(* Logix 5000 project; controller Sucrose_Main Emulate 5570 rev 20.12; software revision 20.01; part 17 of 30 *)
(* tags used below, declared in another part *)
   Alarm_ACK_Master_Timer : TIMER;
   DO_E22_5 : ALIAS FOR FLX_E22:5:O;   // Discrete Output EN2T_FLX 192.168.1.22
   FV230602_AOI : QSI_Flow_Valve;   // FV-23-06-02 PRE FILTER TRAIN 2 INLET LOW POINT DRAIN VALVE
   FV230603_AOI : QSI_Flow_Valve;   // FV-23-06-03 PRE FILTER TRAIN 2 INLET LOW POINT DRAIN VALVE
   FV230604_AOI : QSI_Flow_Valve;   // FV-23-06-04 PRE FILTER TRAIN 2 OUTLET LOW POINT DRAIN VALVE
   FV230605_AOI : QSI_Flow_Valve;   // FV-23-06-05 PRE FILTER TRAIN 2 OUTLET LOW POINT DRAIN VALVE
   FV230607_AOI : QSI_Flow_Valve;   // FV-23-06-07 LOW POINT DRAIN VALVE
   FV230609_AOI : QSI_Flow_Valve;   // FV-23-06-09 FINAL FILTER TRAIN 2 INLET LOW POINT DRAIN VALVE
   FV230610_AOI : QSI_Flow_Valve;   // FV-23-06-10 FINAL FILTER TRAIN 2 INLET LOW POINT DRAIN VALVE
   FV230611_AOI : QSI_Flow_Valve;   // FV-23-06-11 FINAL FILTER TRAIN 2 OUTLET LOW POINT DRAIN VALVE
   FV230612_AOI : QSI_Flow_Valve;   // FV-23-06-12 FINAL FILTER TRAIN 2 OUTLET LOW POINT DRAIN VALVE
   Sucrose_MM_Enable : BOOL;
   SucroseCIP_FILTRATION_REMOTE : CIP_REMOTE;
   SucroseFiltration : Area_Program;
(* FiltrationArea_EN2T_IO_Discrete_DO_E22_5, continued *)

ROUTINE _03_FV230602   (* ladder *)
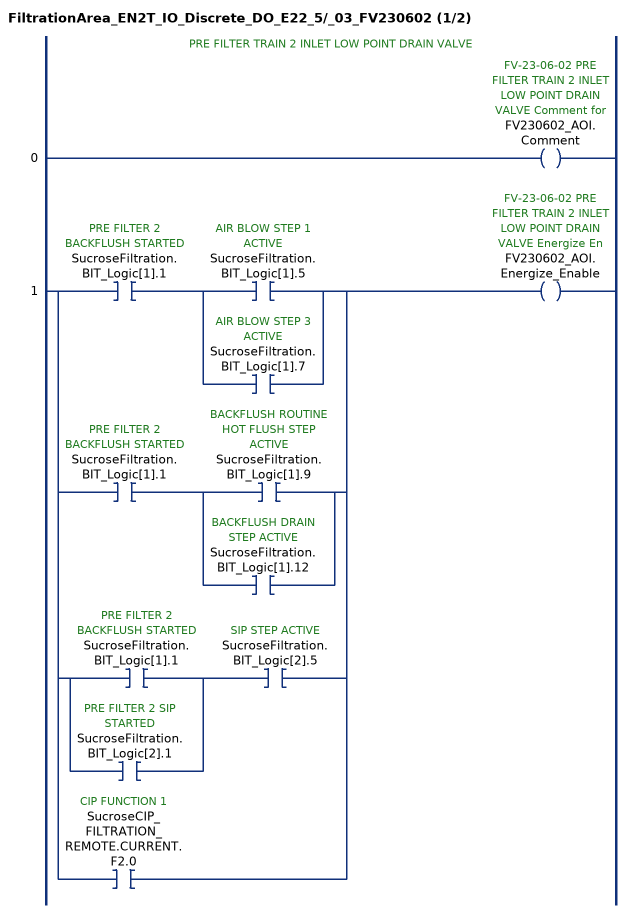
   // PRE FILTER TRAIN 2 INLET LOW POINT DRAIN VALVE
   0: OTE(FV230602_AOI.Comment);
   1: [XIC(SucroseFiltration.BIT_Logic[1].1) [XIC(SucroseFiltration.BIT_Logic[1].5) ,XIC(SucroseFiltration.BIT_Logic[1].7) ] ,XIC(SucroseFiltration.BIT_Logic[1].1) [XIC(SucroseFiltration.BIT_Logic[1].9) ,XIC(SucroseFiltration.BIT_Logic[1].12) ] ,[XIC(SucroseFiltration.BIT_Logic[1].1) ,XIC(SucroseFiltration.BIT_Logic[2].1) ] XIC(SucroseFiltration.BIT_Logic[2].5) ,XIC(SucroseCIP_FILTRATION_REMOTE.CURRENT.F2.0) ]OTE(FV230602_AOI.Energize_Enable);
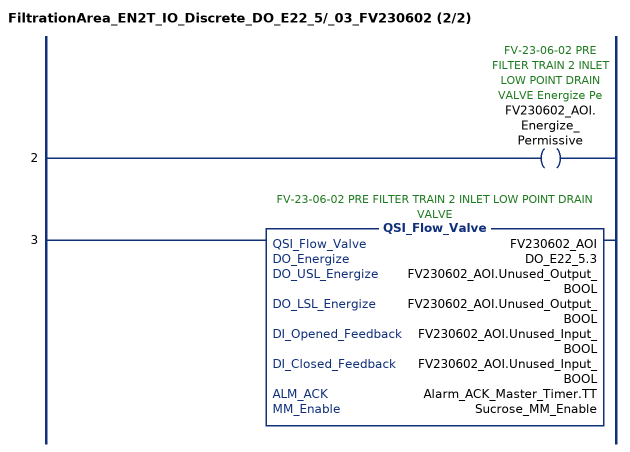
   2: OTE(FV230602_AOI.Energize_Permissive);
   3: QSI_Flow_Valve(FV230602_AOI,DO_E22_5.3,FV230602_AOI.Unused_Output_BOOL,FV230602_AOI.Unused_Output_BOOL,FV230602_AOI.Unused_Input_BOOL,FV230602_AOI.Unused_Input_BOOL,Alarm_ACK_Master_Timer.TT,Sucrose_MM_Enable);
END_ROUTINE

ROUTINE _04_FV230603   (* ladder *)
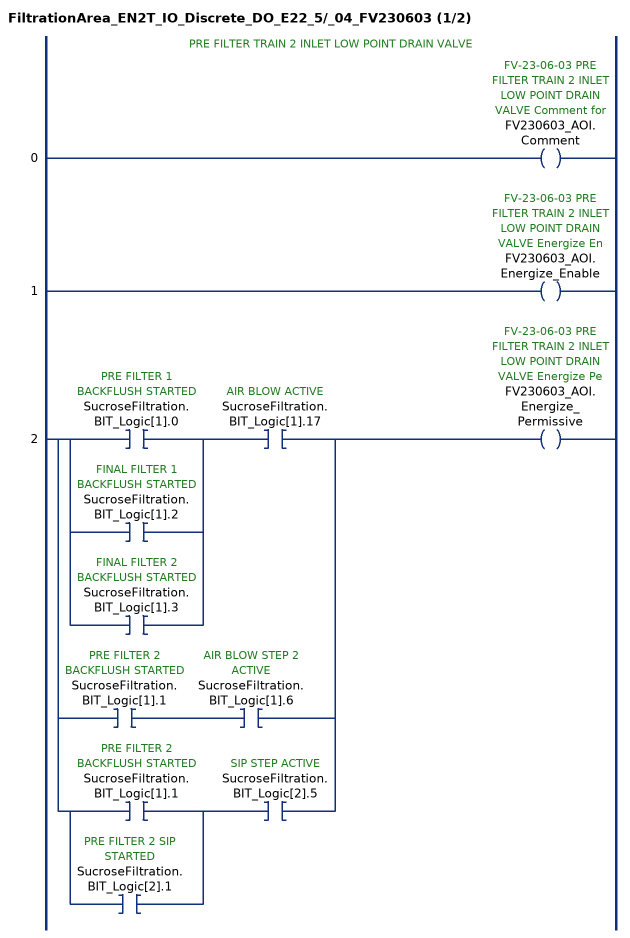
   // PRE FILTER TRAIN 2 INLET LOW POINT DRAIN VALVE
   0: OTE(FV230603_AOI.Comment);
   1: OTE(FV230603_AOI.Energize_Enable);
   2: [[XIC(SucroseFiltration.BIT_Logic[1].0) ,XIC(SucroseFiltration.BIT_Logic[1].2) ,XIC(SucroseFiltration.BIT_Logic[1].3) ] XIC(SucroseFiltration.BIT_Logic[1].17) ,XIC(SucroseFiltration.BIT_Logic[1].1) XIC(SucroseFiltration.BIT_Logic[1].6) ,[XIC(SucroseFiltration.BIT_Logic[1].1) ,XIC(SucroseFiltration.BIT_Logic[2].1) ] XIC(SucroseFiltration.BIT_Logic[2].5) ]OTE(FV230603_AOI.Energize_Permissive);
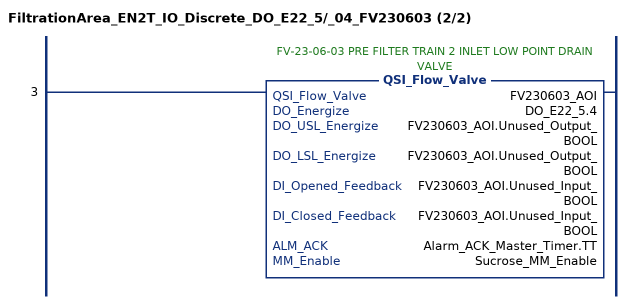
   3: QSI_Flow_Valve(FV230603_AOI,DO_E22_5.4,FV230603_AOI.Unused_Output_BOOL,FV230603_AOI.Unused_Output_BOOL,FV230603_AOI.Unused_Input_BOOL,FV230603_AOI.Unused_Input_BOOL,Alarm_ACK_Master_Timer.TT,Sucrose_MM_Enable);
END_ROUTINE

ROUTINE _05_FV230604   (* ladder *)
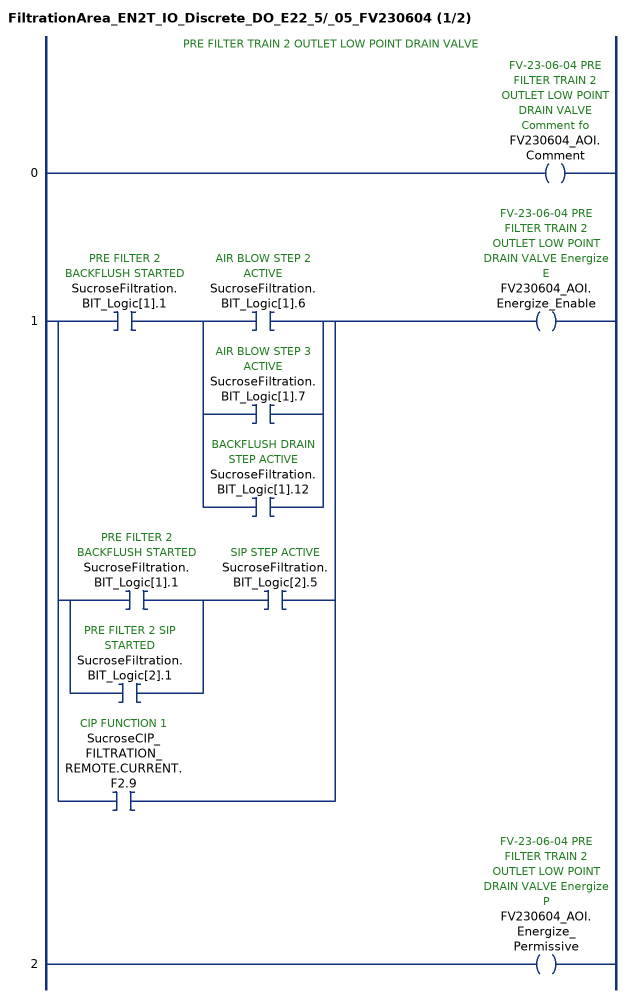
   // PRE FILTER TRAIN 2 OUTLET LOW POINT DRAIN VALVE
   0: OTE(FV230604_AOI.Comment);
   1: [XIC(SucroseFiltration.BIT_Logic[1].1) [XIC(SucroseFiltration.BIT_Logic[1].6) ,XIC(SucroseFiltration.BIT_Logic[1].7) ,XIC(SucroseFiltration.BIT_Logic[1].12) ] ,[XIC(SucroseFiltration.BIT_Logic[1].1) ,XIC(SucroseFiltration.BIT_Logic[2].1) ] XIC(SucroseFiltration.BIT_Logic[2].5) ,XIC(SucroseCIP_FILTRATION_REMOTE.CURRENT.F2.9) ]OTE(FV230604_AOI.Energize_Enable);
   2: OTE(FV230604_AOI.Energize_Permissive);
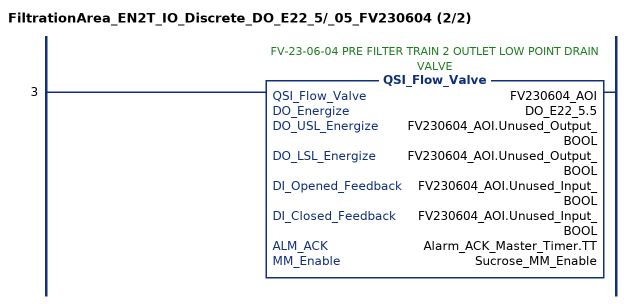
   3: QSI_Flow_Valve(FV230604_AOI,DO_E22_5.5,FV230604_AOI.Unused_Output_BOOL,FV230604_AOI.Unused_Output_BOOL,FV230604_AOI.Unused_Input_BOOL,FV230604_AOI.Unused_Input_BOOL,Alarm_ACK_Master_Timer.TT,Sucrose_MM_Enable);
END_ROUTINE

ROUTINE _06_FV230605   (* ladder *)
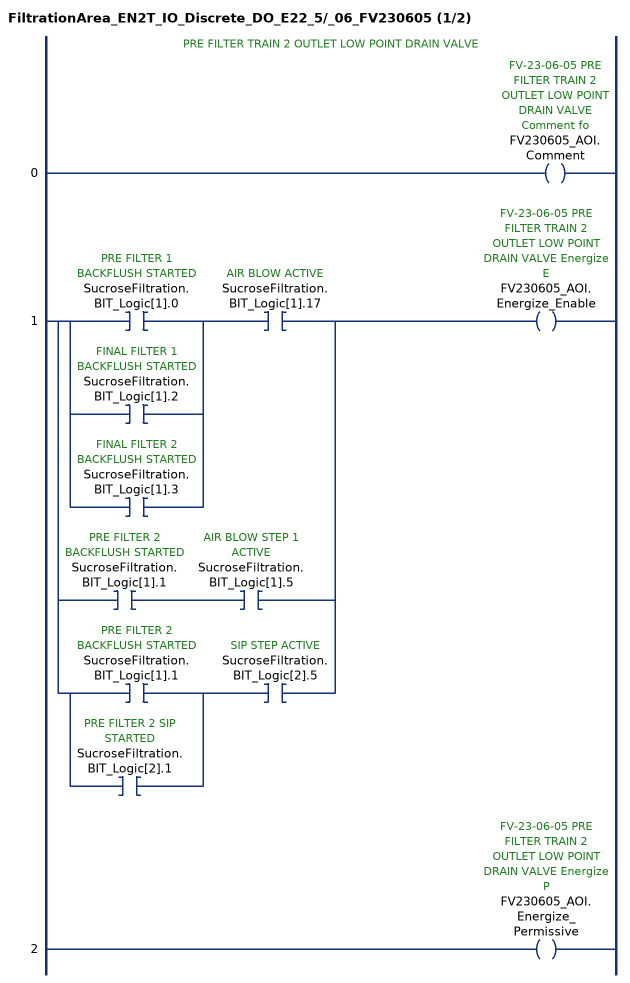
   // PRE FILTER TRAIN 2 OUTLET LOW POINT DRAIN VALVE
   0: OTE(FV230605_AOI.Comment);
   1: [[XIC(SucroseFiltration.BIT_Logic[1].0) ,XIC(SucroseFiltration.BIT_Logic[1].2) ,XIC(SucroseFiltration.BIT_Logic[1].3) ] XIC(SucroseFiltration.BIT_Logic[1].17) ,XIC(SucroseFiltration.BIT_Logic[1].1) XIC(SucroseFiltration.BIT_Logic[1].5) ,[XIC(SucroseFiltration.BIT_Logic[1].1) ,XIC(SucroseFiltration.BIT_Logic[2].1) ] XIC(SucroseFiltration.BIT_Logic[2].5) ]OTE(FV230605_AOI.Energize_Enable);
   2: OTE(FV230605_AOI.Energize_Permissive);
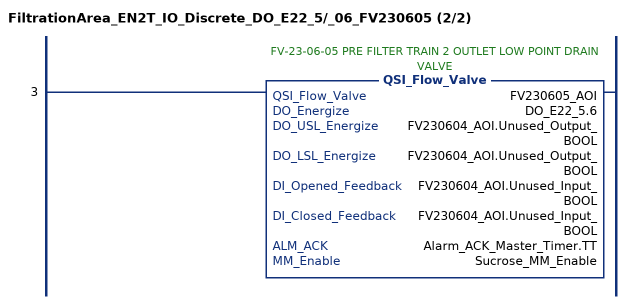
   3: QSI_Flow_Valve(FV230605_AOI,DO_E22_5.6,FV230604_AOI.Unused_Output_BOOL,FV230604_AOI.Unused_Output_BOOL,FV230604_AOI.Unused_Input_BOOL,FV230604_AOI.Unused_Input_BOOL,Alarm_ACK_Master_Timer.TT,Sucrose_MM_Enable);
END_ROUTINE

ROUTINE _07_FV230607   (* ladder *)
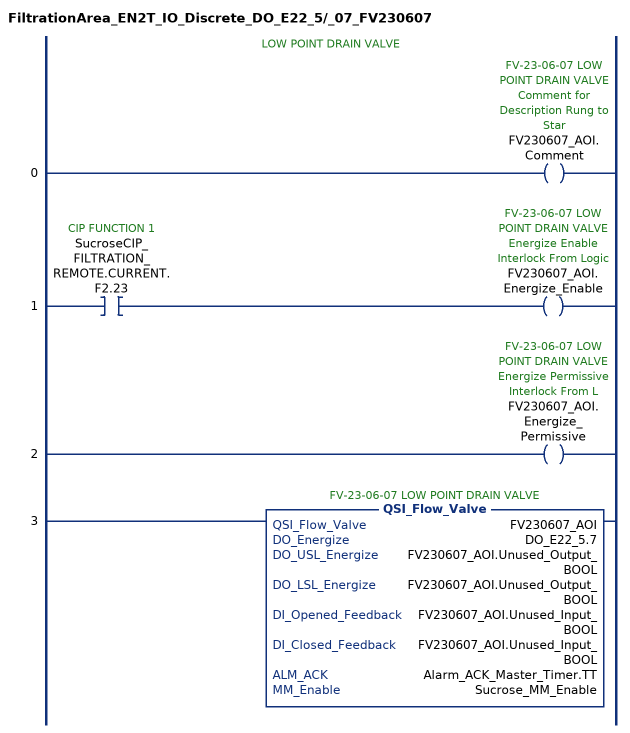
   // LOW POINT DRAIN VALVE
   0: OTE(FV230607_AOI.Comment);
   1: XIC(SucroseCIP_FILTRATION_REMOTE.CURRENT.F2.23)OTE(FV230607_AOI.Energize_Enable);
   2: OTE(FV230607_AOI.Energize_Permissive);
   3: QSI_Flow_Valve(FV230607_AOI,DO_E22_5.7,FV230607_AOI.Unused_Output_BOOL,FV230607_AOI.Unused_Output_BOOL,FV230607_AOI.Unused_Input_BOOL,FV230607_AOI.Unused_Input_BOOL,Alarm_ACK_Master_Timer.TT,Sucrose_MM_Enable);
END_ROUTINE

ROUTINE _08_FV230609   (* ladder *)
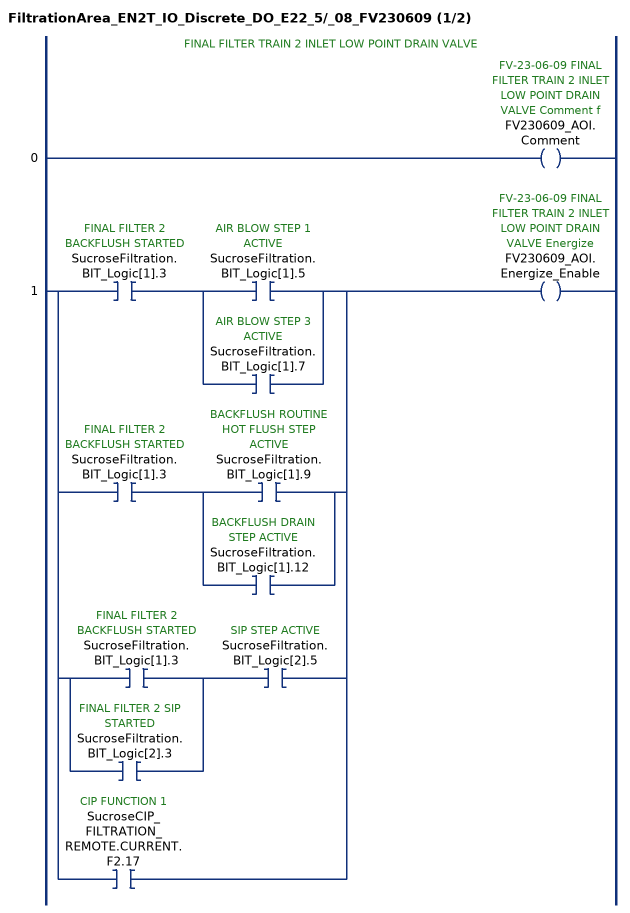
   // FINAL FILTER TRAIN 2 INLET LOW POINT DRAIN VALVE
   0: OTE(FV230609_AOI.Comment);
   1: [XIC(SucroseFiltration.BIT_Logic[1].3) [XIC(SucroseFiltration.BIT_Logic[1].5) ,XIC(SucroseFiltration.BIT_Logic[1].7) ] ,XIC(SucroseFiltration.BIT_Logic[1].3) [XIC(SucroseFiltration.BIT_Logic[1].9) ,XIC(SucroseFiltration.BIT_Logic[1].12) ] ,[XIC(SucroseFiltration.BIT_Logic[1].3) ,XIC(SucroseFiltration.BIT_Logic[2].3) ] XIC(SucroseFiltration.BIT_Logic[2].5) ,XIC(SucroseCIP_FILTRATION_REMOTE.CURRENT.F2.17) ]OTE(FV230609_AOI.Energize_Enable);
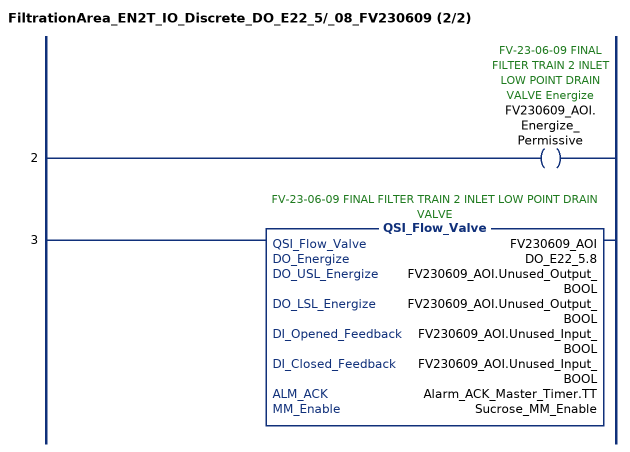
   2: OTE(FV230609_AOI.Energize_Permissive);
   3: QSI_Flow_Valve(FV230609_AOI,DO_E22_5.8,FV230609_AOI.Unused_Output_BOOL,FV230609_AOI.Unused_Output_BOOL,FV230609_AOI.Unused_Input_BOOL,FV230609_AOI.Unused_Input_BOOL,Alarm_ACK_Master_Timer.TT,Sucrose_MM_Enable);
END_ROUTINE

ROUTINE _09_FV230610   (* ladder *)
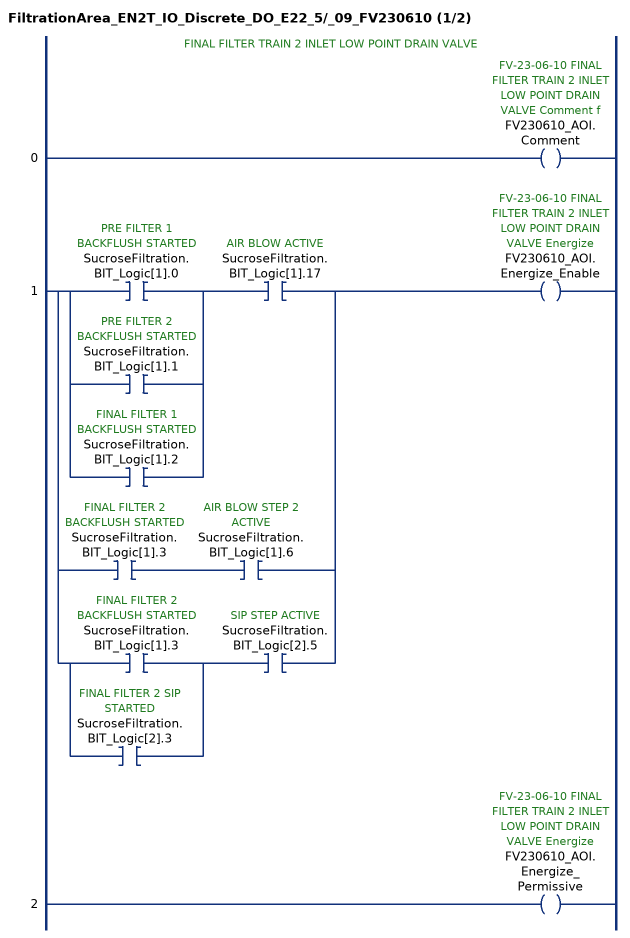
   // FINAL FILTER TRAIN 2 INLET LOW POINT DRAIN VALVE
   0: OTE(FV230610_AOI.Comment);
   1: [[XIC(SucroseFiltration.BIT_Logic[1].0) ,XIC(SucroseFiltration.BIT_Logic[1].1) ,XIC(SucroseFiltration.BIT_Logic[1].2) ] XIC(SucroseFiltration.BIT_Logic[1].17) ,XIC(SucroseFiltration.BIT_Logic[1].3) XIC(SucroseFiltration.BIT_Logic[1].6) ,[XIC(SucroseFiltration.BIT_Logic[1].3) ,XIC(SucroseFiltration.BIT_Logic[2].3) ] XIC(SucroseFiltration.BIT_Logic[2].5) ]OTE(FV230610_AOI.Energize_Enable);
   2: OTE(FV230610_AOI.Energize_Permissive);
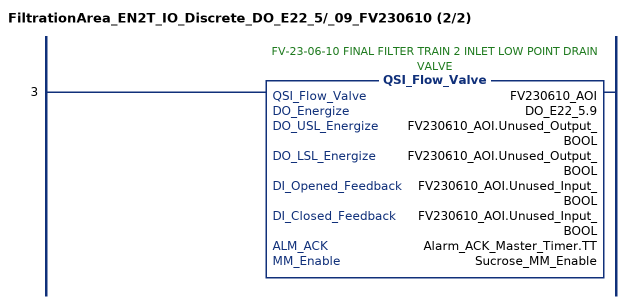
   3: QSI_Flow_Valve(FV230610_AOI,DO_E22_5.9,FV230610_AOI.Unused_Output_BOOL,FV230610_AOI.Unused_Output_BOOL,FV230610_AOI.Unused_Input_BOOL,FV230610_AOI.Unused_Input_BOOL,Alarm_ACK_Master_Timer.TT,Sucrose_MM_Enable);
END_ROUTINE

ROUTINE _10_FV230611   (* ladder *)
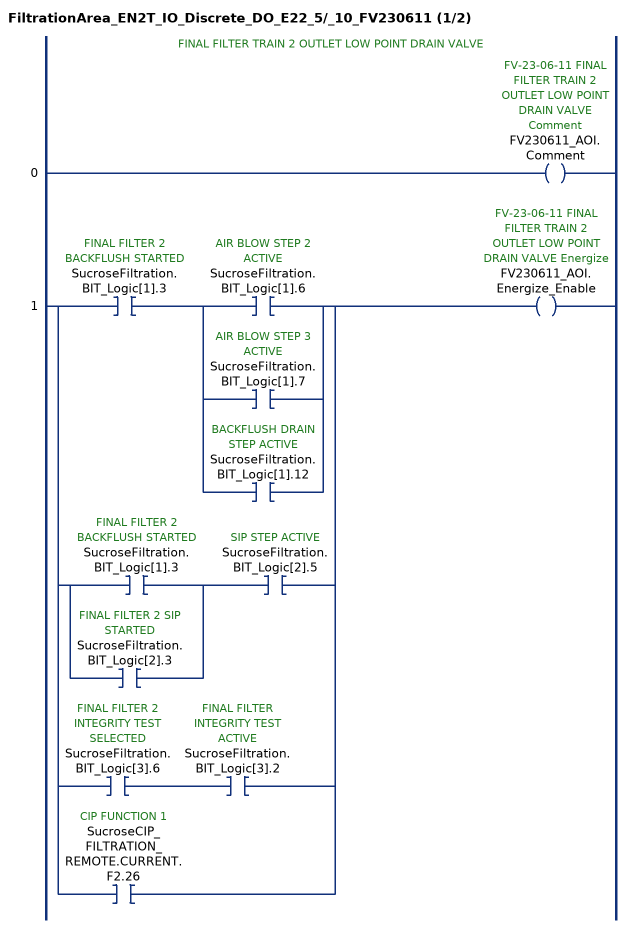
   // FINAL FILTER TRAIN 2 OUTLET LOW POINT DRAIN VALVE
   0: OTE(FV230611_AOI.Comment);
   1: [XIC(SucroseFiltration.BIT_Logic[1].3) [XIC(SucroseFiltration.BIT_Logic[1].6) ,XIC(SucroseFiltration.BIT_Logic[1].7) ,XIC(SucroseFiltration.BIT_Logic[1].12) ] ,[XIC(SucroseFiltration.BIT_Logic[1].3) ,XIC(SucroseFiltration.BIT_Logic[2].3) ] XIC(SucroseFiltration.BIT_Logic[2].5) ,XIC(SucroseFiltration.BIT_Logic[3].6) XIC(SucroseFiltration.BIT_Logic[3].2) ,XIC(SucroseCIP_FILTRATION_REMOTE.CURRENT.F2.26) ]OTE(FV230611_AOI.Energize_Enable);
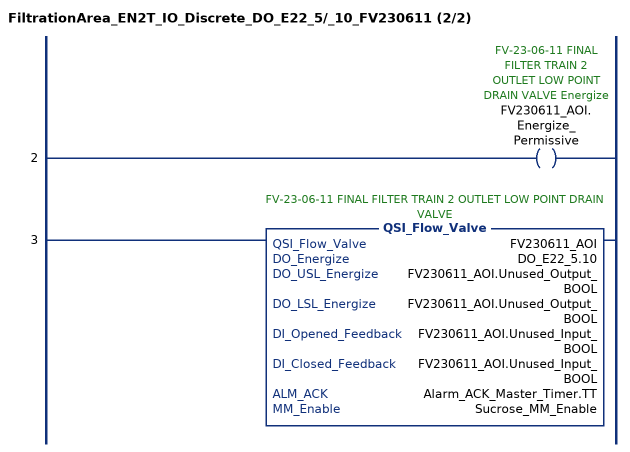
   2: OTE(FV230611_AOI.Energize_Permissive);
   3: QSI_Flow_Valve(FV230611_AOI,DO_E22_5.10,FV230611_AOI.Unused_Output_BOOL,FV230611_AOI.Unused_Output_BOOL,FV230611_AOI.Unused_Input_BOOL,FV230611_AOI.Unused_Input_BOOL,Alarm_ACK_Master_Timer.TT,Sucrose_MM_Enable);
END_ROUTINE

ROUTINE _11_FV230612   (* ladder *)
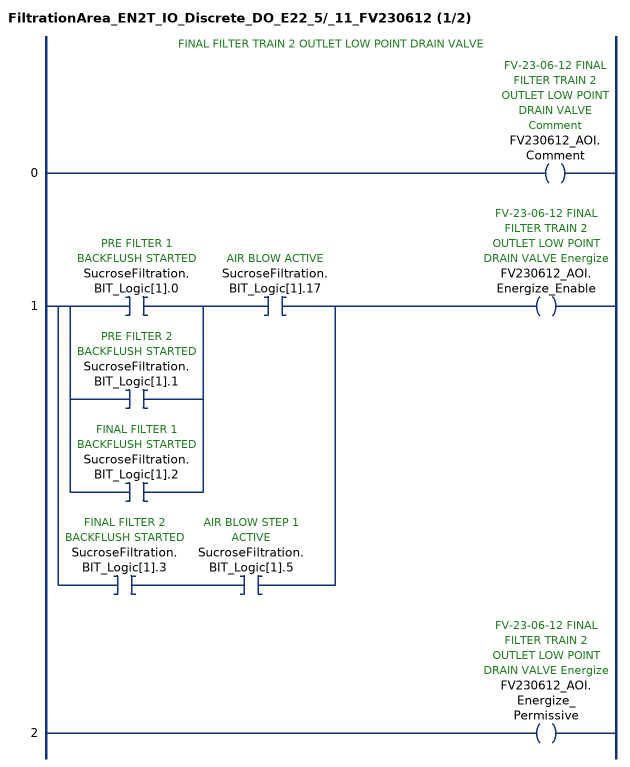
   // FINAL FILTER TRAIN 2 OUTLET LOW POINT DRAIN VALVE
   0: OTE(FV230612_AOI.Comment);
   1: [[XIC(SucroseFiltration.BIT_Logic[1].0) ,XIC(SucroseFiltration.BIT_Logic[1].1) ,XIC(SucroseFiltration.BIT_Logic[1].2) ] XIC(SucroseFiltration.BIT_Logic[1].17) ,XIC(SucroseFiltration.BIT_Logic[1].3) XIC(SucroseFiltration.BIT_Logic[1].5) ]OTE(FV230612_AOI.Energize_Enable);
   2: OTE(FV230612_AOI.Energize_Permissive);
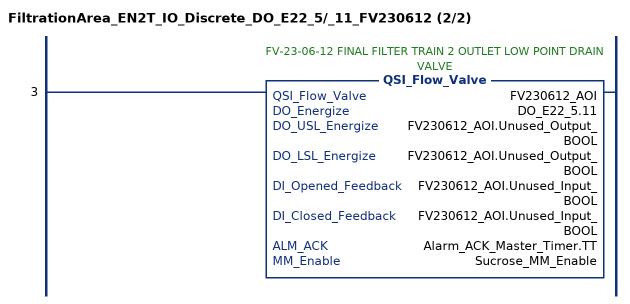
   3: QSI_Flow_Valve(FV230612_AOI,DO_E22_5.11,FV230612_AOI.Unused_Output_BOOL,FV230612_AOI.Unused_Output_BOOL,FV230612_AOI.Unused_Input_BOOL,FV230612_AOI.Unused_Input_BOOL,Alarm_ACK_Master_Timer.TT,Sucrose_MM_Enable);
END_ROUTINE

ROUTINE MainRoutine   (* ladder *)
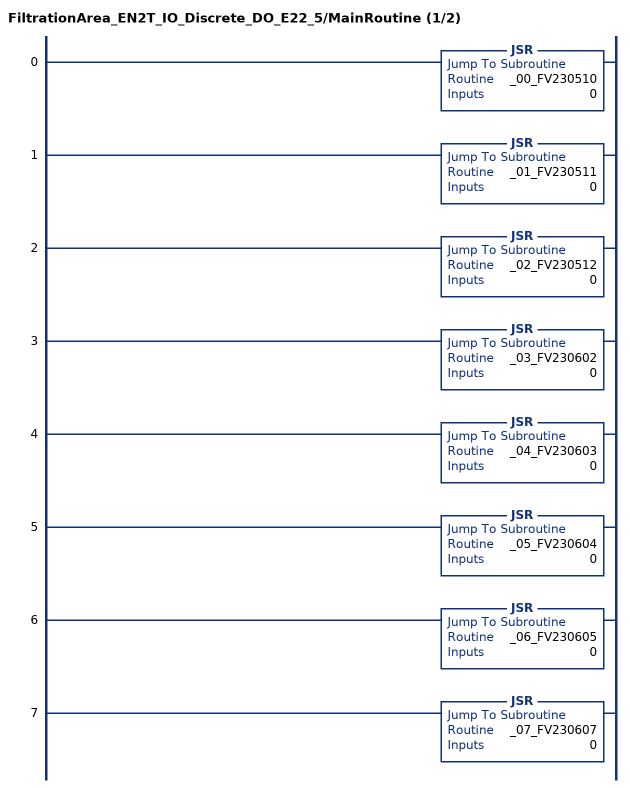
   0: JSR(_00_FV230510,0);
   1: JSR(_01_FV230511,0);
   2: JSR(_02_FV230512,0);
   3: JSR(_03_FV230602,0);
   4: JSR(_04_FV230603,0);
   5: JSR(_05_FV230604,0);
   6: JSR(_06_FV230605,0);
   7: JSR(_07_FV230607,0);
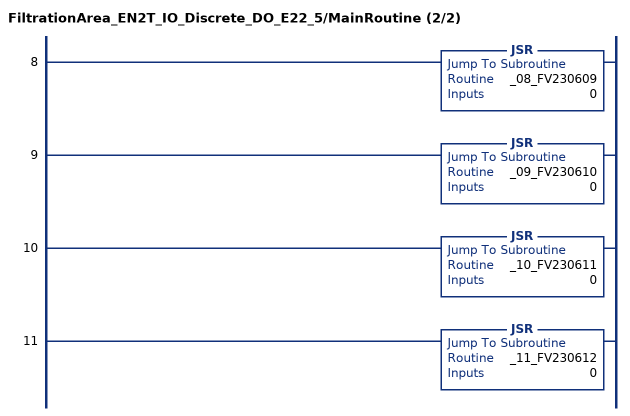
   8: JSR(_08_FV230609,0);
   9: JSR(_09_FV230610,0);
   10: JSR(_10_FV230611,0);
   11: JSR(_11_FV230612,0);
END_ROUTINE
END_PROGRAM
